PROGRAM FactoryIO_ModbusTCP
VAR
	fb_FactoryIO_ModbusTCP : FB_FactoryIO_ModbusTCP;

END_VAR

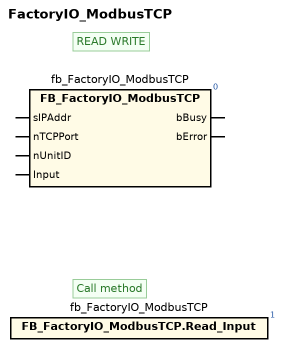
// READ WRITE
fb_FactoryIO_ModbusTCP();
// Call method
fb_FactoryIO_ModbusTCP.Read_Input();

END_PROGRAM

(* stored: Version 1.1.0.1, ProductVersion 3.1.4024.11
   POU FactoryIO_ModbusTCP: Id {e3a0b526-1f07-43ca-9585-e7d3202c3fc5}, SpecialFunc None *)
